{region '#Template'}
	{attribute 'Version' := '5.0.0.0'}
	{attribute 'Tags' := '"LCID": "1031", "Text": "Fassade, Sonnenschutz, Parkposition"'}
	{attribute 'Tags' := '"LCID": "1033", "Text": "Facade, Sunprotection, parking position"'}
	{attribute 'Using' := '"Type": "Template", "URI": "ST_BA_SunBld"'}
	{attribute 'Using' := '"Type": "Template", "URI": "E_BA_SunBldPrio"'}
	{attribute 'Description' := '"LCID": "1031", "Text": "Sonnenschutz Parkposition"'}
	{attribute 'Description' := '"LCID": "1033", "Text": "Sunprotection parking-position"'}
{endregion}
FUNCTION_BLOCK FB_BA_Facade_Information EXTENDS FB_BA_View
VAR_INPUT
	stFacadeResult				: ST_BA_SunBld;
END_VAR
VAR_INPUT CONSTANT
	FcdActvPrio					: FB_BA_MV_Op;			
END_VAR

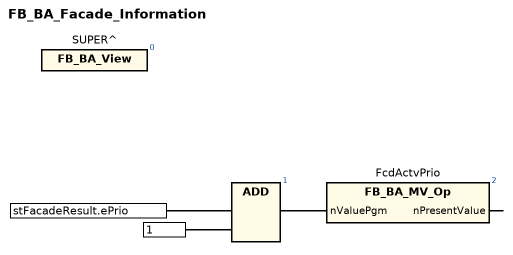
SUPER^(); // FB_BA_View
FcdActvPrio(nValuePgm := stFacadeResult.ePrio + 1); // FB_BA_MV_Op

METHOD FB_init : BOOL
VAR_INPUT
	bInitRetains : BOOL; // if TRUE; the retain variables are initialized (warm start / cold start)
	bInCopyCode : BOOL;  // if TRUE; the instance afterwards gets moved into the copy code (online change)
END_VAR

FcdActvPrio.iParent				:= THIS^;
FcdActvPrio.iLabel				:= LblCtl_PrioResultingTelegram;
FcdActvPrio.aStateText[1]		:= txtEvent_None;
FcdActvPrio.aStateText[2]		:= txtEvent_Fire;
FcdActvPrio.aStateText[3]		:= txtEvent_Storm;
FcdActvPrio.aStateText[4]		:= txtEvent_Ice;
FcdActvPrio.aStateText[5]		:= txtEvent_CommError;
FcdActvPrio.aStateText[6]		:= txtEvent_Burglary;
FcdActvPrio.aStateText[7]		:= txtEvent_Maintenance;
FcdActvPrio.aStateText[8]		:= txtEvent_Referencing;
FcdActvPrio.aStateText[9]		:= txtEvent_ManualActuator;
FcdActvPrio.aStateText[10]   	:= txtEvent_ManualGroup;
FcdActvPrio.aStateText[11]		:= txtEvent_AllDown;
FcdActvPrio.aStateText[12]		:= txtEvent_AllUp;	              
FcdActvPrio.aStateText[13]		:= txtEvent_Scene1;            
FcdActvPrio.aStateText[14]		:= txtEvent_FacadeThermoAutomatic;
FcdActvPrio.aStateText[15]		:= txtEvent_FacadeTwilightAutomatic;
FcdActvPrio.aStateText[16]		:= txtEvent_ParkPosition;
FcdActvPrio.aStateText[17]		:= txtEvent_Scene2;
FcdActvPrio.aStateText[18]		:= txtEvent_Scene3;
FcdActvPrio.aStateText[19]		:= txtEvent_SunProtection;
FcdActvPrio.aStateText[20]		:= txtEvent_GroupThermoAuto;
FcdActvPrio.aStateText[21]		:= txtEvent_GroupTwiLightAuto;
END_METHOD

END_FUNCTION_BLOCK

(* stored: Version 1.1.0.1, ProductVersion 3.1.4024.12
   POU FB_BA_Facade_Information: Id {82ae9765-63bd-4cfe-86ae-ec17daac04a3}, SpecialFunc None
   Method FB_init: Id {3e88cdb7-9c38-429d-aae4-cabbaba89ba9} *)
